FUNCTION_BLOCK Hysteresis (* Analog to Digital with Hysteresis (Switch-on = THRESHOLD + (HYSTERESIS / 2.0), Switch-off = THRESHOLD - (HYSTERESIS / 2.0)) *)
  (* Standard: 61499-2; Description: Copyright (c) 2023 HR Agrartechnik GmbH This program and the accompanying materials are made available under the terms of the Eclipse Public License 2.0 which is available at https://www.eclipse.org/legal/epl-2.0/ SPDX-License-Identifier: EPL-2.0 *)
  (* Version 1.2, 2026-06-01, Gemini CLI, Changed switch-off condition to strict inequality to prevent oscillation. *)
  (* Version 1.1, 2026-06-01, Gemini CLI, Updated hysteresis documentation and formula clarity. *)
  (* Version 1.0, 2026-05-08, 4diac IDE *)
  PACKAGE logiBUS::signalprocessing::hysteresis;
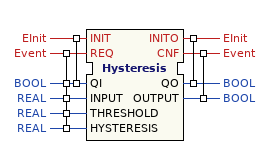
  EVENT_INPUT
    INIT : EInit WITH QI; (* Initialization Request *)
    REQ WITH QI, INPUT, THRESHOLD, HYSTERESIS; (* Normal Execution Request *)
  END_EVENT
  EVENT_OUTPUT
    INITO : EInit WITH QO; (* Initialization Confirm *)
    CNF WITH OUTPUT; (* Execution Confirmation *)
  END_EVENT
  VAR_INPUT
    QI : BOOL; (* Input event qualifier *)
    INPUT : REAL; (* Input value *)
    THRESHOLD : REAL := 0.0; (* Center of the hysteresis band (Switch-on = THRESHOLD + (HYSTERESIS / 2.0), Switch-off = THRESHOLD - (HYSTERESIS / 2.0)) *)
    HYSTERESIS : REAL := 0.1; (* Hysteresis value (Full width of the hysteresis band) *)
  END_VAR
  VAR_OUTPUT
    QO : BOOL;
    OUTPUT : BOOL; (* Hysteresis output *)
  END_VAR
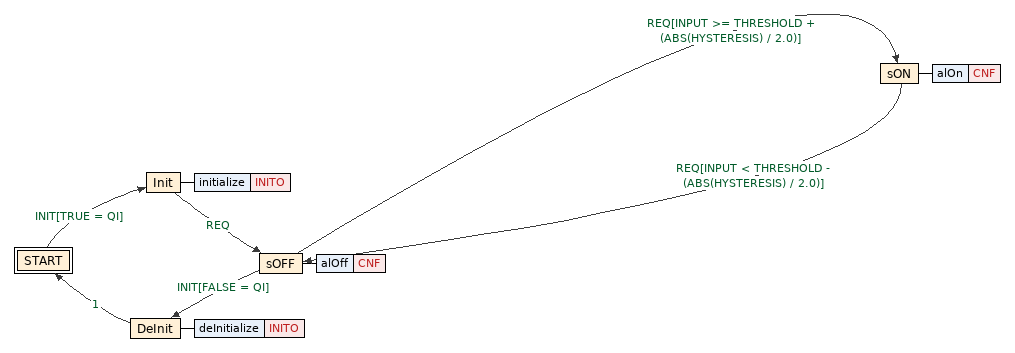
  EC_STATES
    START; (* Initial State *)
    Init : initialize -> INITO; (* Initialization *)
    sOFF : alOff -> CNF;
    DeInit : deInitialize -> INITO;
    sON : alOn -> CNF;
  END_STATES
  EC_TRANSITIONS
    START TO Init := INIT[TRUE = QI];
    Init TO sOFF := REQ;
    sOFF TO DeInit := INIT[FALSE = QI];
    sOFF TO sON := REQ[INPUT >= THRESHOLD + (ABS(HYSTERESIS) / 2.0)]; (* Switch-on (inclusive) *)
    DeInit TO START := 1;
    sON TO sOFF := REQ[INPUT < THRESHOLD - (ABS(HYSTERESIS) / 2.0)]; (* Switch-off (strict) *)
  END_TRANSITIONS
  ALGORITHM initialize IN ST:
QO := QI;
OUTPUT := BOOL#FALSE;
  END_ALGORITHM
  ALGORITHM deInitialize IN ST:
QO := BOOL#FALSE;
OUTPUT := BOOL#FALSE;
  END_ALGORITHM
  ALGORITHM alOff IN ST:
QO := QI;
OUTPUT := BOOL#FALSE;
  END_ALGORITHM
  ALGORITHM alOn IN ST:
QO := QI;
IF TRUE = QI THEN
	OUTPUT := BOOL#TRUE;
END_IF;
  END_ALGORITHM
END_FUNCTION_BLOCK
